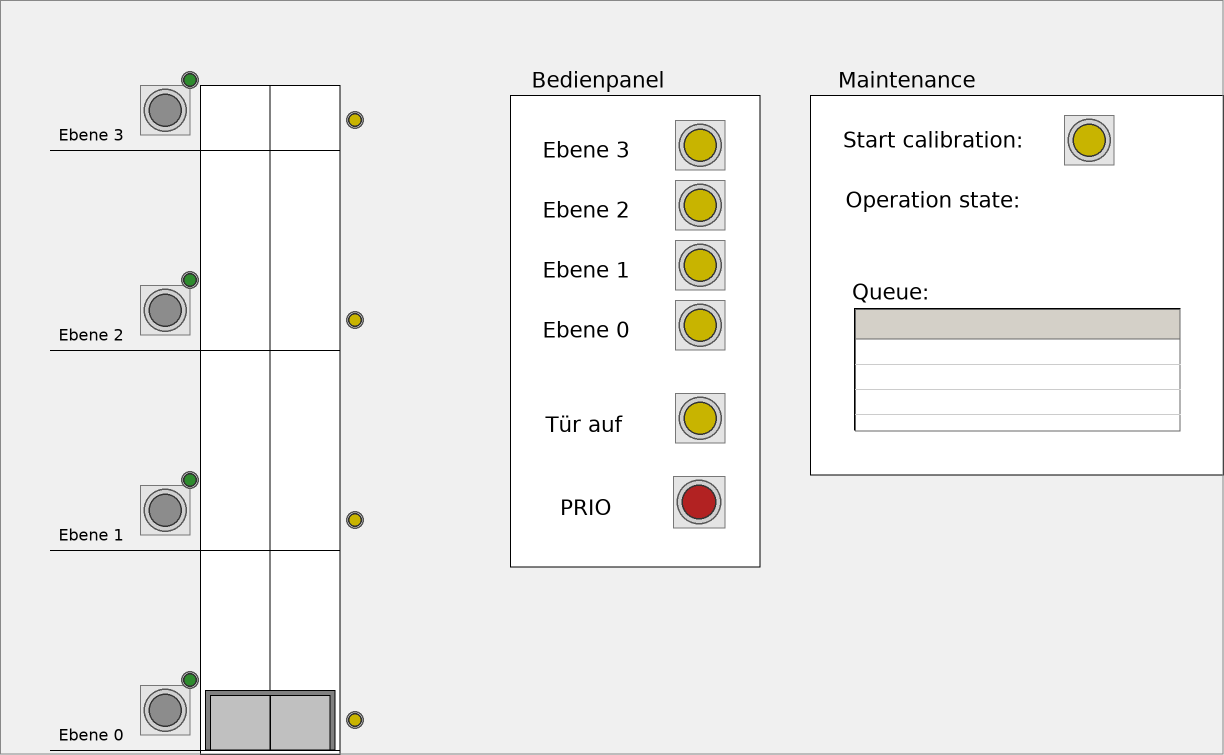
VISUALIZATION Visualization  // 1224x755
    RoundedRectangle (510,95 250x472)
    Lamp1 (345,710 20x20), variable: MAIN.elevatorCtrl.bProxSensors[1], style: Lamp-Lamp1-Yellow
    Rectangle (200,85 140x670)
    Lamp1 (345,510 20x20), variable: MAIN.elevatorCtrl.bProxSensors[2], style: Lamp-Lamp1-Yellow
    Lamp1 (345,310 20x20), variable: MAIN.elevatorCtrl.bProxSensors[3], style: Lamp-Lamp1-Yellow
    Lamp1 (345,110 20x20), variable: MAIN.elevatorCtrl.bProxSensors[4], style: Lamp-Lamp1-Yellow
    Line (50,750) (340,750)
    Line (50,550) (340,550)
    Line (50,350) (340,350)
    Line (50,150) (340,150)
    Label (50,120 82x30), "Ebene 3"
    Label (50,320 82x30), "Ebene 2"
    Label (50,520 82x30), "Ebene 1"
    Label (50,720 82x30), "Ebene 0"
    Rectangle (205,690 130x60)
        p2738717112: -MAIN.liftSim.nLiftPos/2
    Rectangle (210,695 120x55)
        p2738717112: -MAIN.liftSim.nLiftPos/2
    Rectangle (210,695 60x55)
        p874137650: -MAIN.liftSim.nDoorPos/2
        p2738717112: -MAIN.liftSim.nLiftPos/2
    Rectangle (270,695 60x55)
        p2738717112: -MAIN.liftSim.nLiftPos/2
        p3528305787: MAIN.liftSim.nDoorPos/2
    PushSwitch (140,285 50x50), variable: bCallLift[3], behaviour: TAP, style: Switch-PushSwitch-Gray
    PushSwitch (140,85 50x50), variable: bCallLift[4], behaviour: TAP, style: Switch-PushSwitch-Gray
    PushSwitch (140,485 50x50), variable: bCallLift[2], behaviour: TAP, style: Switch-PushSwitch-Gray
    PushSwitch (140,685 50x50), variable: bCallLift[1], behaviour: TAP, style: Switch-PushSwitch-Gray
    PushSwitch (675,120 50x50), variable: bCallLift_Panel[4], behaviour: TAP, style: Switch-PushSwitch-Yellow
    Label (545,135 82x30), "Ebene 3"
    Label (545,195 82x30), "Ebene 2"
    PushSwitch (675,180 50x50), variable: bCallLift_Panel[3], behaviour: TAP, style: Switch-PushSwitch-Yellow
    PushSwitch (675,240 50x50), variable: bCallLift_Panel[2], behaviour: TAP, style: Switch-PushSwitch-Yellow
    Label (545,255 82x30), "Ebene 1"
    Label (545,315 82x30), "Ebene 0"
    PushSwitch (675,300 50x50), variable: bCallLift_Panel[1], behaviour: TAP, style: Switch-PushSwitch-Yellow
    Label (541,408 86x33), "Tür auf"
    Label (498,65 200x30), "Bedienpanel"
    RoundedRectangle (810,95 414x380)
    Label (807,65 200x30), "Maintenance"
    Label (850,125 166x30), "Start calibration:"
    PushSwitch (1064,115 50x50), variable: bInit, behaviour: TAP, style: Switch-PushSwitch-Yellow
    Label (843,185 180x30), "Operation state:"
    Label (843,220 347x40)
    Rectangle (845,219 354x30), text list: 'txt_opMode', text index: MAIN.elevatorCtrl.operationMode
    PushSwitch (675,393 50x50), variable: bOpenDoor, behaviour: TAP, style: Switch-PushSwitch-Yellow
    Rectangle (854,308 326x122)
    Table (855,309 325x122), data array: MAIN.queueLogic.nQueue
        p3854506369: MAIN.queueLogic.nQueue[INDEX]
    Label (843,277 95x30), "Queue:"
    Lamp1 (180,670 20x20), variable: MAIN.queueLogic.bLevelInQueue[1], style: Lamp-Lamp1-Green
    Lamp1 (180,470 20x20), variable: MAIN.queueLogic.bLevelInQueue[2], style: Lamp-Lamp1-Green
    Lamp1 (180,270 20x20), variable: MAIN.queueLogic.bLevelInQueue[3], style: Lamp-Lamp1-Green
    Lamp1 (180,70 20x20), variable: MAIN.queueLogic.bLevelInQueue[4], style: Lamp-Lamp1-Green
    Line (270,690) (270,85)
        p2773130477: -MAIN.liftSim.nLiftPos/2
    Label (543,491 86x33), "PRIO"
    PushSwitch (673,476 52x52), variable: bSetPrio, behaviour: TOGGLE, style: Switch-PushSwitch-Red
END_VISUALIZATION

(* stored: Version 1.1.0.1, ProductVersion 3.1.4024.6
   Visu Visualization: Id {41170220-a534-4e10-8777-e32f5ed0d977} *)
